(*

.. <legal notes>

legal notes
=================
| SPDX-FileCopyrightText: © 2026 Oleksandr Tiutyk <trofimich@gmail.com>
| SPDX-License-Identifier: LGPL-3.0-only
| For details check: LGPL-3.0-only_

.. _LGPL-3.0-only: https://www.gnu.org/licenses/lgpl-3.0.en.html

.. </legal notes>

*)

FUNCTION_BLOCK ABSTRACT Device EXTENDS Core.Object IMPLEMENTS IDevice
VAR
	_Name : WSTRING;
	
	_Parent : IAutomationComponent;
	
	_Enabled : BOOL := TRUE;
	
	_SimulationModeOverride : SIMULATION_MODE_OVERRIDE;
END_VAR

METHOD ABSTRACT Disable
END_METHOD

METHOD ABSTRACT Enable
VAR_INPUT
	includeChildren : BOOL := TRUE;
END_VAR
END_METHOD

{attribute 'monitoring' := 'call'}
PROPERTY FINAL Enabled : BOOL
GET
Enabled := _Enabled;
END_GET
END_PROPERTY

METHOD FB_init : BOOL
VAR_INPUT
	(* if TRUE, the retain variables are initialized (warm start / cold start)*)
	bInitRetains	: BOOL;
	(* if TRUE, the instance afterwards gets moved into the copy code (online change)*)
	bInCopyCode	: BOOL;
	parent : IAutomationComponent;
	name : WSTRING;
END_VAR
_Parent := parent;
_Name := SEL(Core.WideStrings.IsNullOrWhiteSpace(name), name, GetDefaultName());
END_METHOD

METHOD ABSTRACT Initialize : BOOL
END_METHOD

{attribute 'monitoring' := 'call'}
PROPERTY FINAL Name : WSTRING
GET
Name := _Name;
END_GET
END_PROPERTY

{attribute 'monitoring' := 'call'}
PROPERTY FINAL Parent : IAutomationComponent
GET
Parent := _Parent;
END_GET
END_PROPERTY

METHOD SetSimulationModeOverride
VAR_INPUT
	value : SIMULATION_MODE_OVERRIDE;
END_VAR
END_METHOD

{attribute 'monitoring' := 'call'}
PROPERTY FINAL SimulationMode : BOOL
GET
CASE _SimulationModeOverride OF
	SIMULATION_MODE_OVERRIDE.INHERITED:
		SimulationMode := _Parent.SimulationMode;
 	
	SIMULATION_MODE_OVERRIDE.ON:
		SimulationMode := TRUE;
	
	SIMULATION_MODE_OVERRIDE.OFF:
		SimulationMode := FALSE;
END_CASE
END_GET
END_PROPERTY

{attribute 'monitoring' := 'call'}
PROPERTY FINAL SimulationModeOverride : SIMULATION_MODE_OVERRIDE
GET
SimulationModeOverride := _SimulationModeOverride;
END_GET
END_PROPERTY

END_FUNCTION_BLOCK

(* stored: Version 1.1.0.1
   POU Device: Id {f3b4f1f5-d7e8-495b-a404-a87157d5f32f}, SpecialFunc None
   Method Disable: Id {a589d881-30ab-45e0-8243-ebd458820f89}
   Method Enable: Id {25a6d708-22d7-4efa-8813-16fc8241d52a}
   Property Enabled: Id {cf2193ce-5af9-47f7-b767-75a7e05b3149}
   Get Get: Id {ec5c75a6-430a-4018-81a9-b306246e2aeb}
   Method FB_init: Id {6e7d33a1-6d80-43ad-a8d8-899454af5a81}
   Method Initialize: Id {f9c960f5-7e68-42ba-bfa8-19000f1f0084}
   Property Name: Id {5d75ce6c-7303-4356-bdac-c2abe75bfc34}
   Get Get: Id {0a48de5b-eca6-4414-ba3e-f68dae0edc4a}
   Property Parent: Id {9a2a0d18-500c-4856-b3bd-133e8d7de4d2}
   Get Get: Id {5e19e287-9498-42dd-bbfe-2069a9e5105e}
   Method SetSimulationModeOverride: Id {5f49bbb1-2cc6-4576-ac29-53d7da71ae0d}
   Property SimulationMode: Id {9d8291ac-cf17-4d5c-8fae-88749aefade2}
   Get Get: Id {b1008e3c-64f8-46c5-b998-489b78df3ea4}
   Property SimulationModeOverride: Id {9d85b7a1-31f3-4304-8474-17c8363c1a0c}
   Get Get: Id {61ac5dd9-17b7-4a39-85eb-963f627be032} *)
